// TwinCAT 3 PLC project conveyor_plc_project
// ProgramVersion: 3.1.4024.0
// libraries:
//   Tc2_Standard, * (Beckhoff Automation GmbH)
//   Tc2_System, * (Beckhoff Automation GmbH)
//   Tc3_Module, * (Beckhoff Automation GmbH)
// project tree:
//   Conveyor/ FB_Conveyor.TcPOU
//   DUTs/ E_ConveyorState.TcDUT, ST_ConveyorInputs.TcDUT, ST_ConveyorOutputs.TcDUT
//   GVLs/ GVL_IO.TcGVL
//   / PlcTask.TcTTO
//   POUs/ MAIN.TcPOU

CONFIGURATION conveyor_plc_project
    RESOURCE PLC ON TwinCAT3
        TASK PlcTask(INTERVAL := T#10ms, PRIORITY := 20);
        PROGRAM MAIN WITH PlcTask : MAIN;
    END_RESOURCE
END_CONFIGURATION

// ---- DUTs/E_ConveyorState.TcDUT
{attribute 'qualified_only'}
{attribute 'strict'}
TYPE E_ConveyorState :
(
	INIT := 0,
	REQUEST_MOVE	:=1,
	MOVING			:=2,
	STOP			:=3,
	ERROR			:=4
);
END_TYPE

// ---- DUTs/ST_ConveyorInputs.TcDUT
TYPE ST_ConveyorInputs :
STRUCT
	bConveyorIsMoving	:BOOL;
	bConveyorStopped	:BOOL;
	bPartDetected		:BOOL;
	bPartAvailable2Move	:BOOL;
	bRobInSpace			:BOOL;
END_STRUCT
END_TYPE

// ---- DUTs/ST_ConveyorOutputs.TcDUT
TYPE ST_ConveyorOutputs :
STRUCT
	bMoveConveyor	:BOOL;
	bStopConveyor	:BOOL;
	bEnableConveyor	:BOOL;
	
END_STRUCT
END_TYPE

// ---- GVLs/GVL_IO.TcGVL
{attribute 'qualified_only'}
VAR_GLOBAL
	Conveyor_Inputs		:ST_ConveyorInputs;
	Conveyor_Outputs	:ST_ConveyorOutputs;
END_VAR

// ---- POUs/MAIN.TcPOU
PROGRAM MAIN
VAR
	fbConveyor	:FB_Conveyor;
END_VAR

fbConveyor(stInput	:= GVL_IO.Conveyor_Inputs, stOutput=>GVL_IO.Conveyor_Outputs);

END_PROGRAM

// ---- Conveyor/FB_Conveyor.TcPOU
FUNCTION_BLOCK FB_Conveyor
VAR_INPUT
	stInput	:ST_ConveyorInputs;
END_VAR
VAR_OUTPUT
	stOutput	:ST_ConveyorOutputs;
END_VAR
VAR
	eActConveyorState	:E_ConveyorState	:= E_ConveyorState.INIT;
	bPartDetected		:BOOL	:=FALSE;
END_VAR

A_ProcessFlow();

ACTION A_ProcessFlow:
CASE eActConveyorState OF 
	E_ConveyorState.INIT:
		// When conveyor part is at the end of the conveyor stop it. robot will clear the part
		IF M_PartDetectedAtEnd() THEN
			eActConveyorState := E_ConveyorState.STOP;
		END_IF
		
		// When part is not at the end, start the conveyor to move 
		IF NOT M_PartDetectedAtEnd()  AND NOT stInput.bRobInSpace THEN
			IF P_GetPart2Move THEN
				eActConveyorState	:= E_ConveyorState.REQUEST_MOVE;
			END_IF
		END_IF
	
		
		
	E_ConveyorState.REQUEST_MOVE:
		stOutput.bMoveConveyor := TRUE;
		eActConveyorState	:= E_ConveyorState.MOVING;
		
		
		
	E_ConveyorState.MOVING:
		IF P_GetConveyorMoving THEN
			// DO Nothing. Wait here until Part is detected
			
		END_IF
		IF M_PartDetectedAtEnd() THEN
			eActConveyorState	:= E_ConveyorState.STOP;
		END_IF
		
		
		
	E_ConveyorState.STOP:
		stOutput.bMoveConveyor := FALSE;
		IF NOT P_GetConveyorMoving THEN
			// DO Nothing
			eActConveyorState	:= E_ConveyorState.INIT;
		ELSE
			eActConveyorState	:= E_ConveyorState.ERROR;
		END_IF
		
		
		
	E_ConveyorState.ERROR:
		// TODO: Wait for Error Handling
		
END_CASE

bPartDetected	:= M_PartDetectedAtEnd();
END_ACTION

METHOD M_PartDetectedAtEnd : BOOL
VAR_INPUT
END_VAR
M_PartDetectedAtEnd := stInput.bPartDetected;
RETURN;
END_METHOD

PROPERTY P_GetConveyorMoving : BOOL
GET
stInput.bConveyorIsMoving := stOutput.bMoveConveyor;
END_GET
END_PROPERTY

PROPERTY P_GetPart2Move : BOOL
GET
P_GetPart2Move := GVL_IO.Conveyor_Inputs.bPartAvailable2Move;
END_GET
END_PROPERTY

END_FUNCTION_BLOCK
